{attribute 'GeneratedUsingTerminal: EK1122-0000-0018'}
{attribute addProperty BoxType "EK1122-0000-0018"}
{attribute addProperty Id "Beckhoff_ELM9xxxsub_EK1100EK1100_AB5A94672"}
{attribute addProperty CRC "644013717"}
{attribute addProperty Size "2"}
TYPE Beckhoff_ELM9xxxEK1122_2662DE95 EXTENDS EK1122_AB5A9467 :
STRUCT
	{attribute addProperty Name "Beckhoff_ELM9xxxsub_EK1100"}
	{attribute addProperty PreviousPort "Beckhoff ELM9xxxEK1122 : D"}
	Beckhoff_ELM9xxxsub_EK1100 : EK1100_AB5A9467;
END_STRUCT
END_TYPE

(* stored: Version 1.2.0.0, ProductVersion 3.1.4024.9
   DUT Beckhoff_ELM9xxxEK1122_2662DE95: Id {d78a9d6b-ced9-4eb5-87f5-de5db2bcff84} *)
